// TIA Portal V20 export
TYPE "TypeAxisRd"
   STRUCT
      TargetPos : DInt;   // target position [mm/10]
      CalibratePos : DInt;   // calibrated position [mm/10]
      RefPosToBoard : DInt;   // reference position to board [mm/10]
      SetCalibratePos : Bool;   // set calibrated position
      ManModeActive : Bool;   // manual mode active
      ManPlus : Bool;   // manual plus
      ManMinus : Bool;   // manual minus
      ManRefRun : Bool;   // manual reference run
   END_STRUCT;
END_TYPE
